TYPE T_Port : UINT; END_TYPE

(* stored: Version 1.1.0.1, ProductVersion 3.1.4024.15
   DUT T_Port: Id {e25cf913-34e0-0a62-05c2-18d76ac59ca3} *)
